PROGRAM MovementTypeSelector
VAR
	fbGcode : FB_Movement_Gcode;
	fbHome : FB_HbotHome;
	fbXbox : FB_Movement_Xbox;
	limx : BOOL;
	limy : BOOL;
	
	caseswitch : (none, home, gcode, teach, vision, error);
END_VAR

CASE caseswitch OF
	none:
	fbGcode(bExecute := FALSE);
	fbXbox(bExecute := FALSE);
	fbHome(bExecute := FALSE, StepperA := GVL.StepperReferenceA, StepperB := GVL.StepperReferenceB,limitSwitchX := GVL.LimitSwitchMidLeft, limitSwitchY := GVL.LimitSwitchBotLeft);
		(* 20230712: Decoupling from HMI, for now clicking on Xbox Controller's Select btn goes to Teach *)
		IF tcXbox.xBoxController.P_Buttons.bB_Button THEN
			caseswitch := teach;
		END_IF
		
		(* Home first before going into Teach If you do not, it will take its current location as "0" although it technically doesnt matter for now*)
		(*IF TcXbox.xBoxController.P_Buttons.bA_Button THEN 
			caseswitch := home;
		END_IF*) //UNCOMMENT AFTER LIMIT SWITCHES ARE READY YOU RETARD 
		
	home:
		fbHome(bExecute := TRUE, StepperA := GVL.StepperReferenceA, StepperB := GVL.StepperReferenceB,
			limitSwitchX := GVL.LimitSwitchMidLeft, limitSwitchY := GVL.LimitSwitchBotLeft);
		IF fbHome.bError THEN
			caseswitch := error;
		ELSIF fbHome.bDone THEN
			fbHome(bExecute := FALSE, StepperA := GVL.StepperReferenceA, StepperB := GVL.StepperReferenceB,
			limitSwitchX := GVL.LimitSwitchMidLeft, limitSwitchY := GVL.LimitSwitchBotLeft);
			caseswitch := none;
		END_IF
		
	gcode:
		fbGcode(bExecute := TRUE);
		IF fbGcode.bFinished AND NOT fbGcode.initial.Q THEN
			caseswitch := none;
		END_IF
		
	teach:
		fbXbox(bExecute := TRUE);

	Error:
		caseswitch := None;
		
END_CASE

END_PROGRAM

(* stored: Version 1.1.0.1, ProductVersion 3.1.4024.12
   POU MovementTypeSelector: Id {05a34db7-57c4-4ffe-a0a1-689688bc2c16}, SpecialFunc None *)
